FUNCTION_BLOCK SUBL_94 (* 94-variable local group subscriber *)
  (* Standard: 61499-2 *)
  (* Version 1.0, 21-03-12, GASR, Universidade do Estado de Santa Catarina *)
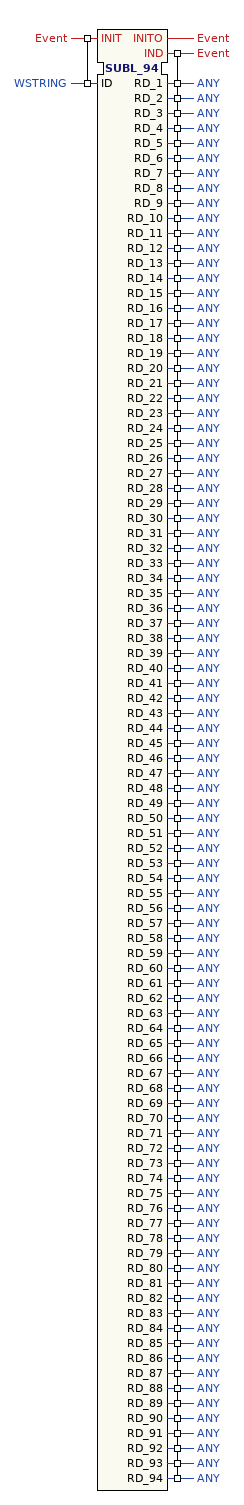
  EVENT_INPUT
    INIT WITH ID; (* Service Initialization *)
  END_EVENT
  EVENT_OUTPUT
    INITO; (* Initialization Confirm *)
    IND WITH RD_1, RD_2, RD_3, RD_4, RD_5, RD_6, RD_7, RD_8, RD_9, RD_10, RD_11, RD_12, RD_13, RD_14, RD_15, RD_16, RD_17, RD_18, RD_19, RD_20, RD_21, RD_22, RD_23, RD_24, RD_25, RD_26, RD_27, RD_28, RD_29, RD_30, RD_31, RD_32, RD_33, RD_34, RD_35, RD_36, RD_37, RD_38, RD_39, RD_40, RD_41, RD_42, RD_43, RD_44, RD_45, RD_46, RD_47, RD_48, RD_49, RD_50, RD_51, RD_52, RD_53, RD_54, RD_55, RD_56, RD_57, RD_58, RD_59, RD_60, RD_61, RD_62, RD_63, RD_64, RD_65, RD_66, RD_67, RD_68, RD_69, RD_70, RD_71, RD_72, RD_73, RD_74, RD_75, RD_76, RD_77, RD_78, RD_79, RD_80, RD_81, RD_82, RD_83, RD_84, RD_85, RD_86, RD_87, RD_88, RD_89, RD_90, RD_91, RD_92, RD_93, RD_94; (* Service Indication *)
  END_EVENT
  VAR_INPUT
    ID : WSTRING; (* Default id is the FB instance name *)
  END_VAR
  VAR_OUTPUT
    RD_1 : ANY; (* pos *)
    RD_2 : ANY; (* current_tool *)
    RD_3 : ANY; (* setup.Its_secplane.position.location.coordinates *)
    RD_4 : ANY; (* round_hole.its_id *)
    RD_5 : ANY; (* its_workpiece.its_id *)
    RD_6 : ANY; (* its_operations.its_id LIST - the list is concatenated in one string *)
    RD_7 : ANY; (* feature_placement.name *)
    RD_8 : ANY; (* feature_placement.location.name *)
    RD_9 : ANY; (* feature_placement.location.coordinates *)
    RD_10 : ANY; (* feature_placement.axis.its_id *)
    RD_11 : ANY; (* feature_placement.axis.direction_ratios *)
    RD_12 : ANY; (* feature_placement.ref_direction.its_id *)
    RD_13 : ANY; (* feature_placement.ref_direction_ratios *)
    RD_14 : ANY; (* depth.name *)
    RD_15 : ANY; (* depth.postion.name *)
    RD_16 : ANY; (* depth.position.location.name *)
    RD_17 : ANY; (* depth.position.location.coordinates *)
    RD_18 : ANY; (* depth.position.axis.its_id *)
    RD_19 : ANY; (* depth.position.axis.direction_ratios *)
    RD_20 : ANY; (* depth.position.ref_direction.its_id *)
    RD_21 : ANY; (* depth.position.ref_direction_ratios *)
    RD_22 : ANY; (* diameter *)
    RD_23 : ANY; (* diameter.theoretical_size *)
    RD_24 : ANY; (* diameter.implicit_tolerance *)
    RD_25 : ANY; (* diameter.{vector}, vector = {upper_limit, lower_limit, significant_digits} or {deviation,grade,its_fitting_type} *)
    RD_26 : ANY; (* change_in_diameter, "diameter_taper" or "angle_taper" *)
    RD_27 : ANY; (* change_in_diameter.theoretical_size *)
    RD_28 : ANY; (* change_in_diameter.implicit_tolerance *)
    RD_29 : ANY; (* change_in_diameter.{vector}, vector = {upper_limit, lower_limit, significant_digits} or {deviation,grade,its_fitting_type} *)
    RD_30 : ANY; (* bottom_condition, "through_bottom_condition" or ... *)
    RD_31 : ANY; (* bottom_condition.theoretical_size *)
    RD_32 : ANY; (* bottom_condition.implicit_tolerance *)
    RD_33 : ANY; (* bottom_condition.{vector}, vector = {upper_limit, lower_limit, significant_digits} or {deviation,grade,its_fitting_type} *)
    RD_34 : ANY; (* drilling.its_id *)
    RD_35 : ANY; (* its_toolpath.its_list *)
    RD_36 : ANY; (* its_tool_direction *)
    RD_37 : ANY; (* retract_plane *)
    RD_38 : ANY; (* start_point.name *)
    RD_39 : ANY; (* start_point.coordinates *)
    RD_40 : ANY; (* its_tool.its_id *)
    RD_41 : ANY; (* its_tool.its_tool_body.dimension.diameter *)
    RD_42 : ANY; (* its_tool.its_tool_body.dimension.tool_tip_half_angle *)
    RD_43 : ANY; (* its_tool.its_tool_body.dimension.tool_circumference_angle *)
    RD_44 : ANY; (* its_tool.its_tool_body.dimension.cutting_edge_lenght *)
    RD_45 : ANY; (* its_tool.its_tool_body.dimension.edge_radius *)
    RD_46 : ANY; (* its_tool.its_tool_body.dimension.edge_center_vertical *)
    RD_47 : ANY; (* its_tool.its_tool_body.dimension.edge_center_horizontal *)
    RD_48 : ANY; (* its_tool.its_tool_body.number_of_teeth *)
    RD_49 : ANY; (* its_tool.its_tool_body.hand_of_cut *)
    RD_50 : ANY; (* its_tool.its_tool_body.coolant_through *)
    RD_51 : ANY; (* its_tool.its_tool_body.pilot_length *)
    RD_52 : ANY; (* its_tool.its_tool_body.{other_tool_body_parameter} *)
    RD_53 : ANY; (* its_tool.its_cutting_edge.tool_offset_length *)
    RD_54 : ANY; (* its_tool.its_cutting_edge.its_material.standard_identifier *)
    RD_55 : ANY; (* its_tool.its_cutting_edge.its_material.material_identifier *)
    RD_56 : ANY; (* its_tool.its_cutting_edge.its_material.material_property.{list_of_parameters} *)
    RD_57 : ANY; (* its_tool.its_cutting_edge.its_technological_data.cutting_angle *)
    RD_58 : ANY; (* its_tool.its_cutting_edge.its_technological_data.free_angle *)
    RD_59 : ANY; (* its_tool.its_cutting_edge.its_technological_data.aux_angle *)
    RD_60 : ANY; (* its_tool.its_cutting_edge.expected_tool_life *)
    RD_61 : ANY; (* its_tool.its_cutting_edge.its_technology.feedrate *)
    RD_62 : ANY; (* its_tool.its_cutting_edge.its_technology.feedrate_reference *)
    RD_63 : ANY; (* its_tool.its_cutting_edge.its_technology.cutspeed *)
    RD_64 : ANY; (* its_tool.its_cutting_edge.its_technology.spindle *)
    RD_65 : ANY; (* its_tool.its_cutting_edge.its_technology.feedrate_per_tooth *)
    RD_66 : ANY; (* its_tool.its_cutting_edge.its_technology.sincronize_spindle_with_feed *)
    RD_67 : ANY; (* its_tool.its_cutting_edge.its_technology.inhibit_feedrate_override *)
    RD_68 : ANY; (* its_tool.its_cutting_edge.its_technology.inhibit_spindle_override *)
    RD_69 : ANY; (* its_tool.its_cutting_edge.its_technology.its_adaptive_control *)
    RD_70 : ANY; (* its_tool.overall_assembly_length *)
    RD_71 : ANY; (* its_tool.direction_for_spindle_orientation.its_id *)
    RD_72 : ANY; (* its_tool.direction_for_spindle_orientation.direction_ratios *)
    RD_73 : ANY; (* its_tool.tool_holder_diameter_for_spindle_orientation *)
    RD_74 : ANY; (* its_technology.feedrate *)
    RD_75 : ANY; (* its_technology.feedrate_reference *)
    RD_76 : ANY; (* its_technology.cutspeed *)
    RD_77 : ANY; (* its_technology.spindle *)
    RD_78 : ANY; (* its_technology.feedrate_per_tooth *)
    RD_79 : ANY; (* its_technology.sincronize_spindle_with_feed *)
    RD_80 : ANY; (* its_technology.inhibit_feedrate_override *)
    RD_81 : ANY; (* its_technology.inhibit_spindle_override *)
    RD_82 : ANY; (* its_technology.its_adaptive_control *)
    RD_83 : ANY; (* its_machine_functions.coolant *)
    RD_84 : ANY; (* its_machine_functions.coolant_pressure *)
    RD_85 : ANY; (* its_machine_functions.mist *)
    RD_86 : ANY; (* its_machine_functions.through_spindle_coolant *)
    RD_87 : ANY; (* its_machine_functions.through_pressure *)
    RD_88 : ANY; (* its_machine_functions.axis_clamping *)
    RD_89 : ANY; (* its_machine_functions.chip_removal *)
    RD_90 : ANY; (* its_machine_functions.oriented_spindle_stop.its_id *)
    RD_91 : ANY; (* its_machine_functions.oriented_spindle_stop.direction_ratios *)
    RD_92 : ANY; (* its_machine_functions.its_process_model.ini_data_file *)
    RD_93 : ANY; (* its_machine_functions.its_process_model.its_type *)
    RD_94 : ANY; (* its_machine_functions.other_functions *)
  END_VAR
  SERVICE PUBL_105/SUBL_105 (* Data publication service *)
    SEQUENCE normal_establishment
      PUBL_105.INIT(ID) -> PUBL_105.INITO();
      SUBL_105.INIT(ID) -> SUBL_105.INITO();
    END_SEQUENCE
    SEQUENCE normal_data_transfer
      PUBL_105.REQ(SD_1,SD_2,SD_3,SD_4,SD_5,SD_6,SD_7,SD_8,SD_9,SD_10,SD_11,SD_12,SD_13,SD_14,SD_15,SD_16,SD_17,SD_18,SD_19,SD_20,SD_21,SD_22,SD_23,SD_24,SD_25,SD_26,SD_27,SD_28,SD_29,SD_30,SD_31,SD_32,SD_33,SD_34,SD_35,SD_36,SD_37,SD_38,SD_39,SD_40,SD_41,SD_42,SD_43,SD_44,SD_45,SD_46,SD_47,SD_48,SD_49,SD_50,SD_51,SD_52,SD_53,SD_54,SD_55,SD_56,SD_57,SD_58,SD_59,SD_60,SD_61,SD_62,SD_63,SD_64,SD_65,SD_66,SD_67,SD_68,SD_69,SD_70,SD_71,SD_72,SD_73,SD_74,SD_75,SD_76,SD_77,SD_78,SD_79,SD_80,SD_81,SD_82,SD_83,SD_84,SD_85,SD_86,SD_87,SD_88,SD_89,SD_90,SD_91,SD_92,SD_93,SD_94,SD_95,SD_96,SD_97,SD_98,SD_99,SD_100,SD_101,SD_102,SD_103,SD_104,SD_105) -> Subl_105.IND(RD_1,RD_2,RD_3,RD_4,RD_5,RD_6,RD_7,RD_8,RD_9,RD_10,RD_11,RD_12,RD_13,RD_14,RD_15,RD_16,RD_17,RD_18,RD_19,RD_20,RD_21,RD_22,RD_23,RD_24,RD_25,RD_26,RD_27,RD_28,RD_29,RD_30,RD_31,RD_32,RD_33,RD_34,RD_35,RD_36,RD_37,RD_38,RD_39,RD_40,RD_41,RD_42,RD_43,RD_44,RD_45,RD_46,RD_47,RD_48,RD_49,RD_50,RD_51,RD_52,RD_53,RD_54,RD_55,RD_56,RD_57,RD_58,RD_59,RD_60,RD_61,RD_62,RD_63,RD_64,RD_65,RD_66,RD_67,RD_68,RD_69,RD_70,RD_71,RD_72,RD_73,RD_74,RD_75,RD_76,RD_77,RD_78,RD_79,RD_80,RD_81,RD_82,RD_83,RD_84,RD_85,RD_86,RD_87,RD_88,RD_89,RD_90,RD_91,RD_92,RD_93,RD_94,RD_95,RD_96,RD_97,RD_98,RD_99,RD_100,RD_101,RD_102,RD_103,RD_104,RD_105);
    END_SEQUENCE
  END_SERVICE
END_FUNCTION_BLOCK
